Staubli VAL3: Communication.pgx

public program Communication(jointRx& x_jJointRxSend[], jointRx& x_jJointRxRecv[])
  local num l_nDataSend[6]
  local num l_nDataRecv[6]
begin

  //==========双向通讯通道，两个机器人控制器能相互发送和接受数据==========
  //清理Socket缓存，用来接收和发送数据，防止残留数据的干扰
  clearBuffer(sClient)

  //发送指令和数据到服务器，请求数据
  //先解析数据为数组再发送数据
  call jointToArray(x_jJointRxSend,l_nDataSend)
  sioSet(sClient,l_nDataSend)

  //先接受数据再解析为关节位置
  sioGet(sClient,l_nDataRecv)
  call arrayToJoint(l_nDataRecv,x_jJointRxRecv)

end
